// SIMATIC S7-200 project (STEP 7-Micro/WIN), CPU 222 REL 02.01

SYMBOL_TABLE USUARIO1
PARO             I0.0
MARCHA           I0.1
LAMPARA          Q0.0
END_SYMBOL_TABLE

ORGANIZATION_BLOCK PRINCIPAL:OB1
TITLE=COMENTARIOS DEL PROGRAMA
BEGIN
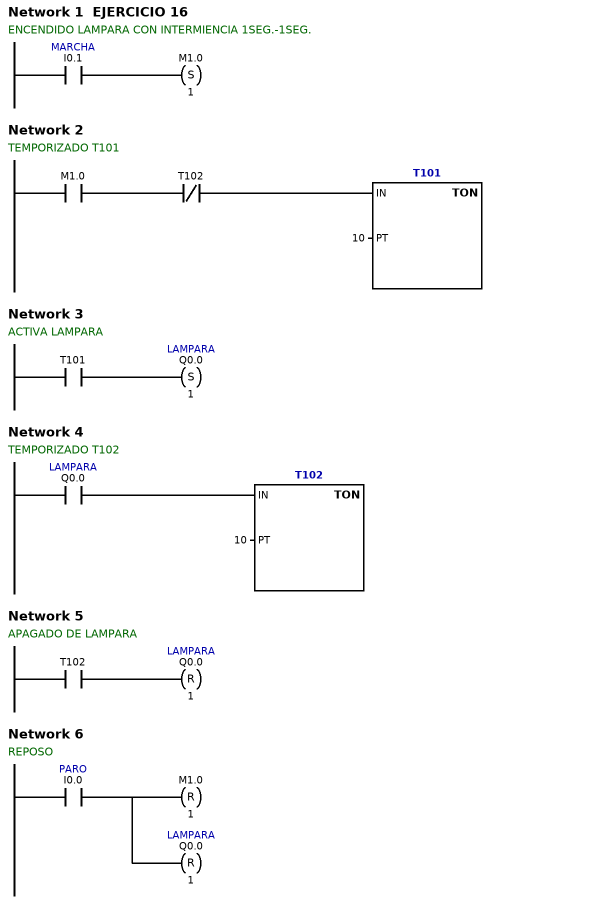
Network 1 // EJERCICIO 16
// ENCENDIDO LAMPARA CON INTERMIENCIA 1SEG.-1SEG.
LD     MARCHA:I0.1
S      M1.0, 1
Network 2
// TEMPORIZADO T101
LD     M1.0
AN     T102
TON    T101, 10
Network 3
// ACTIVA LAMPARA
LD     T101
S      LAMPARA:Q0.0, 1
Network 4
// TEMPORIZADO T102
LD     LAMPARA:Q0.0
TON    T102, 10
Network 5
// APAGADO DE LAMPARA
LD     T102
R      LAMPARA:Q0.0, 1
Network 6
// REPOSO
LD     PARO:I0.0
R      M1.0, 1
R      LAMPARA:Q0.0, 1
END_ORGANIZATION_BLOCK
